// TIA Portal V20 export
// export: Created 2025-12-01T14:57:43.4790721Z, ExportSetting None, DisplayName Totally Integrated Automation Portal, DisplayVersion V20 Update 3, DisplayName TIA Portal Openness, DisplayVersion V20 Update 3, DisplayName TIA Portal Version Control Interface, DisplayVersion V20 Update 3, DisplayName STEP 7 Professional, DisplayVersion V20 Update 3, DisplayName STEP 7 Safety, DisplayVersion V20 Update 2, DisplayName WinCC Basic/Comfort/Advanced, DisplayVersion V20 Update 3, DisplayName WinCC Professional, DisplayVersion V20 Update 3, DisplayName WinCC Unified, DisplayVersion V20 Update 3
FUNCTION "FC503_Borra_FIFO_SCR" : Void   // FC503, LAD
{ S7_Optimized_Access := 'FALSE' }
AUTHOR : TLigero
NAME : 20180425
VERSION : 3.1
// stored: AutoNumber false, SetENOAutomatically false
   VAR_INPUT
      DB_FIFO_Ordenes : UInt;
      Num_Scanner : UInt;   // Numero de scanner sobre el que se realiza la busqueda
      Long_FIFO : UInt;
   END_VAR
   VAR_IN_OUT
      FIFO_OK : Bool;
   END_VAR
   VAR_TEMP
      relleno : Byte;
      retval : Int;
      posicion_actual_N : UInt;
      Registro_Fifo_vacio : "ROUT_Orden_Fifo_Scanner";
   END_VAR
BEGIN

REGION Network 1 (SCL): INICIALIZACION
   REGION INICIALIZACION
       #FIFO_OK := FALSE;
       #relleno := 0;

       #retval:=  FILL(BVAL := #relleno, BLK => #Registro_Fifo_vacio);


   END_REGION

   REGION BUCLE_BORRADO

       FOR #posicion_actual_N := 1 TO #Long_FIFO DO
           // Statement section FOR
           // 
           "FC572_Guardar_Datos_Fifo"(DB_FIFO_Ordenes := #DB_FIFO_Ordenes,
                                      Num_Scanner := #Num_Scanner,
                                      Long_FIFO := #Long_FIFO,
                                      Posicion_FIFO := #posicion_actual_N,
                                      Datos_Scanner_Cruce := #Registro_Fifo_vacio);
       END_FOR;

       #FIFO_OK := TRUE;


       END_REGION
END_REGION
END_FUNCTION
